// TwinCAT 3 PLC project hw_v2
// ProgramVersion: 3.1.4026.22
// libraries:
//   Tc2_Standard, * (Beckhoff Automation GmbH)
//   Tc2_System, * (Beckhoff Automation GmbH)
// project tree:
//   DUTs/ E_State.TcDUT
//   / PlcTask.TcTTO
//   POUs/ FBBTN.TcPOU, FBCOMPARE.TcPOU, FBLED.TcPOU, FBMACHINE.TcPOU, FBUSER.TcPOU, MAIN.TcPOU
// real-time tasks:
//   TASK PlcTask: cycle T#10ms, priority 20, ADS port 350
//   TASK PlcTask1: cycle T#10ms, priority 21, ADS port 351
// I/O:
//   DEVICE Device 1 (EtherCAT), AmsNetId 169.254.56.115.2.1
//     Term 1 (EK1100)
// variable links:
//   (this object) <-> Device 1 (EtherCAT)/Term 1 (EK1100)/Term 2 (EL1008)
//     PlcTask Inputs/MAIN.aBTN[1] <-> Channel 4/Input
//     PlcTask Inputs/MAIN.aBTN[2] <-> Channel 2/Input
//     PlcTask Inputs/MAIN.aBTN[3] <-> Channel 7/Input
//     PlcTask Inputs/MAIN.aBTN[4] <-> Channel 5/Input
//   (this object) <-> Device 1 (EtherCAT)/Term 1 (EK1100)/Term 3 (EL2008)
//     PlcTask Outputs/MAIN.aLED[1] <-> Channel 4/Output
//     PlcTask Outputs/MAIN.aLED[2] <-> Channel 2/Output
//     PlcTask Outputs/MAIN.aLED[3] <-> Channel 7/Output
//     PlcTask Outputs/MAIN.aLED[4] <-> Channel 5/Output
//     PlcTask Outputs/MAIN.aLED[5] <-> Channel 1/Output
//     PlcTask Outputs/MAIN.aLED[6] <-> Channel 3/Output

CONFIGURATION hw_v2
    RESOURCE PLC ON TwinCAT3
        TASK PlcTask(INTERVAL := T#10ms, PRIORITY := 21);
        PROGRAM MAIN WITH PlcTask : MAIN;
    END_RESOURCE
END_CONFIGURATION

// ---- DUTs/E_State.TcDUT
{attribute 'qualified_only'}
{attribute 'strict'}
{attribute 'to_string'}
TYPE E_State :
(
	eSetup,
	eWait,
	eMachine,
	eUser,
	eOutcome,
	eWinner
);
END_TYPE

// ---- POUs/MAIN.TcPOU
PROGRAM MAIN
VAR CONSTANT
	cSTEP_IDLE			: INT := 0;
	cSTEP_PRESS			: INT := 1;
	cSTEP_WAIT			: INT := 10;
	cSTEP_MACHINE		: INT := 20;
	cSTEP_USER			: INT := 30;
	cSTEP_OUTCOME		: INT := 40;
	cSTEP_WINNER		: INT := 50;
	cMaxRound			: INT := 6;
	
	cGreenLED			: INT := 5;
	cRedLED				: INT := 6;
	cBTNtotal			: INT := 4;
	cLEDtotal			: INT := 6;				
END_VAR
VAR
	aBTN AT %I* : ARRAY[1..cBTNtotal] OF BOOL;
	aLED AT %Q* : ARRAY[1..cLEDtotal] OF BOOL;
	
	aBTN_OLD : ARRAY[1..cLEDtotal] OF BOOL;
	aBTN_NEW : ARRAY[1..cLEDtotal] OF BOOL;
	
	aMachine : ARRAY[1..cMaxRound] OF INT;
	aUser : ARRAY[1..cMaxRound] OF INT;
	
	bStepChangeOS		: BOOL;
	nStep				: DINT;
	nStepOld			: DINT;
	
	nCurRound 			: INT;
	fbRand 				: DRAND;
	nSeed 				: INT := 100;
	tonTimer 			: TON;
	bTVar 				: BOOL;
	tTimeout 			: TIME := T#2S;
	tTOn 				: TIME := T#1S;
	tTstb 				: TIME := T#2S;
	nBtnPress 			: INT;
	bOK 				: BOOL;
	
	idx 				: INT := 1;
	cnt 				: INT;
	nWinLED 			: INT;
END_VAR

bStepChangeOS := nStep = nStepOld;
nStepOld := nStep;

tonTimer(IN := bTVar, PT := tTimeout);
nSeed := nSeed + 1;

FOR cnt := 1 TO 4 BY 1 DO
	aBTN_OLD[cnt] := aBTN_NEW[cnt];
	aBTN_NEW[cnt] := aBTN[cnt];
	
	IF aBTN[cnt] THEN
		aLED[cnt] := TRUE;
	ELSE
		aLED[CNT] := FALSE;
	END_IF
END_FOR


// State Machine
CASE nStep OF
	(*************************************************************************************)
	cSTEP_IDLE:		// New game setup
		
	nCurRound := 1;
	bOK := FALSE;
	fbRand(Seed:=nSeed);
	
	IF idx <= cMaxRound THEN
		aMachine[idx] := LREAL_TO_INT(fbRand.Num * 100.0) MOD 3 + 1;
		idx := idx + 1;
	ELSE
		idx := 1;
		nStep := cSTEP_WAIT;
	END_IF
	
		
	(*************************************************************************************)	
	cSTEP_WAIT:		// Wait for user input to start
	
	IF ButtonRelease(bBTN_NEW := aBTN_NEW[1], bBTN_OLD := aBTN_OLD[1]) AND aBTN_NEW[2] THEN
	 	bTVar := TRUE;
		tTimeout := tTstb;
		aLED[cGreenLED] := TRUE;
		aLED[cRedLED] := TRUE;
	END_IF	
	
	IF tonTimer.Q THEN
		aLED[cGreenLED] := FALSE;
		aLED[cRedLED] := FALSE;
		bTVar:=FALSE;
		nStep := cSTEP_MACHINE;
	END_IF
	
	(*************************************************************************************)	
	cSTEP_MACHINE:	// Show Pattern
	
	IF idx <= nCurRound THEN
		IF NOT(tonTimer.Q) THEN
			aLED[aMachine[idx]] := TRUE;
			bTVar := TRUE;
			tTimeout := tTOn;
		ELSE
			aLED[aMachine[idx]] := FALSE;
			bTVar := FALSE;
			idx := idx + 1;
		END_IF
	ELSE
		nStep := cSTEP_USER;
		idx := 1;
	END_IF

	(*************************************************************************************)		
	cSTEP_USER:		// Wait user input
	
	IF idx <= nCurRound THEN
		nBtnPress := GetBR();
		IF NOT(nBtnPress = 0) THEN
			aUser[idx] := nBtnPress;
			IF aMachine[idx] = aUser[idx] THEN
				bOK := TRUE;
				idx := idx + 1;
			ELSE
				bOK := FALSE;
				nStep := cSTEP_OUTCOME;
				idx := 1;
			END_IF
		ELSE
			// do nothing
		END_IF
	ELSE
		nStep := cSTEP_OUTCOME;
		idx := 1;
	END_IF
	
	(*************************************************************************************)		
	cSTEP_OUTCOME:	// Compare machine and user
	
	IF bOK  AND nCurRound < cMaxRound THEN
		nStep := cSTEP_MACHINE;
		nCurRound := nCurRound + 1;
		idx := 1;
	ELSE
		nStep := cSTEP_WINNER;
	END_IF

	
	(*************************************************************************************)		
	cSTEP_WINNER:	// Finishes the game
	
	IF bOK THEN
		nWinLED := cGreenLED;
	ELSE
		nWinLED := cRedLED;
	END_IF
			
	IF NOT(tonTimer.Q) THEN
		aLED[nWinLED] := TRUE;
		bTVar := TRUE;
		tTimeout := tTstb;
	ELSE
		aLED[nWinLED] := FALSE;
		bTVar := FALSE;
		nStep := cSTEP_IDLE;
	END_IF
	
END_CASE

METHOD PRIVATE ButtonPress : BOOL
VAR_INPUT
	bBTN_NEW : BOOL;
	bBTN_OLD : BOOL;
END_VAR

VAR_INST
END_VAR
IF bBTN_OLD = FALSE AND bBTN_NEW = TRUE THEN
	ButtonPress := TRUE;
ELSE
	ButtonPress := FALSE;
END_IF
END_METHOD

METHOD ButtonRelease : BOOL
VAR_INPUT
	bBTN_NEW : BOOL;
	bBTN_OLD : BOOL;
END_VAR
IF bBTN_OLD = TRUE AND bBTN_NEW = FALSE THEN
	ButtonRelease := TRUE;
ELSE
	ButtonRelease := FALSE;
END_IF
END_METHOD

METHOD GetBP : INT
VAR_INPUT
END_VAR
VAR
	loop : int;
END_VAR
FOR loop := 1 TO 4 BY 1 DO
	IF ButtonPress(bBTN_NEW:=aBTN_NEW[loop], bBTN_OLD:=aBTN_OLD[loop]) THEN
		GetBP := loop;
		RETURN;
	ELSE
		GetBP := 0;
	END_IF
END_FOR
END_METHOD

METHOD GetBR : INT
VAR_INPUT
END_VAR
VAR
	loop : INT;
END_VAR
FOR loop := 1 TO 4 BY 1 DO
	IF ButtonRelease(bBTN_NEW := aBTN_NEW[loop], bBTN_OLD := aBTN_OLD[loop]) THEN
		GetBR := loop;
		RETURN;
	ELSE
		GetBR := 0;
	END_IF
END_FOR
END_METHOD

METHOD GetButton : INT
VAR_INPUT
END_VAR
VAR
	loop : INT;
END_VAR
FOR loop := 1 TO 4 BY 1 DO
	IF ButtonPress(bBTN_NEW := aBTN_NEW[loop], bBTN_OLD :=aBTN_OLD[loop]) THEN
		GetButton := loop;
	ELSE
		GetButton := 0;
	END_IF
END_FOR
END_METHOD

END_PROGRAM

// ---- POUs/FBBTN.TcPOU
FUNCTION_BLOCK FBBTN
VAR_INPUT
	bOLD : BOOL;
	bNEW : BOOL;
END_VAR
VAR_OUTPUT
	bOUT : BOOL;
END_VAR
VAR
END_VAR

IF bOLD = FALSE AND bNEW = TRUE THEN
	bOUT := TRUE;
ELSE
	bOUT := FALSE;
END_IF

bOLD := bNEW;

END_FUNCTION_BLOCK

// ---- POUs/FBCOMPARE.TcPOU
FUNCTION_BLOCK FBCOMPARE
VAR_INPUT
END_VAR
VAR_OUTPUT
END_VAR
VAR
END_VAR

END_FUNCTION_BLOCK

// ---- POUs/FBLED.TcPOU
FUNCTION_BLOCK FBLED
VAR_INPUT
END_VAR
VAR_OUTPUT
END_VAR
VAR
END_VAR

END_FUNCTION_BLOCK

// ---- POUs/FBMACHINE.TcPOU
FUNCTION_BLOCK FBMACHINE
VAR_INPUT
END_VAR
VAR_OUTPUT
END_VAR
VAR
END_VAR

END_FUNCTION_BLOCK

// ---- POUs/FBUSER.TcPOU
FUNCTION_BLOCK FBUSER
VAR_INPUT
END_VAR
VAR_OUTPUT
END_VAR
VAR
END_VAR

END_FUNCTION_BLOCK
